// TIA Portal V16 export
// export: Created 2022-11-17T15:49:39.066239Z, ExportSetting WithDefaults, DisplayName Totally Integrated Automation Portal, DisplayVersion V16 Update 6, DisplayName TIA Portal Version Control Interface, DisplayVersion V16 Update 2, DisplayName TIA Portal Openness, DisplayVersion V16 Update 6, DisplayName SINAMICS Startdrive Advanced, DisplayVersion V16 Update 5, DisplayName SINAMICS Startdrive G130, G150, S120, S150, SINAMICS MV, S210, DisplayVersion V16 Update 5, DisplayName SINAMICS Startdrive G110M, G120, G120C, G120D, G120P, G115D, DisplayVersion V16 Update 5, DisplayName STEP 7 Professional, DisplayVersion V16 Update 6, DisplayName STEP 7 Safety, DisplayVersion V16, DisplayName WinCC Advanced, DisplayVersion V16 Update 6
DATA_BLOCK "DB20_DisplaySysdata"   // DB20
{ S7_Optimized_Access := 'FALSE' }
AUTHOR : Robopac
VERSION : 0.0
// stored: AutoNumber false, IsOnlyStoredInLoadMemory false, IsWriteProtectedInAS false
   VAR RETAIN
      dbd0 : DInt := 238;   // Step for encoder spool carriage movement (mm/100) (Display-Sysadata)
      dbw4 : Int := 6;   // Histeresys for spool carriage positioning (mm) (Display-Sysdata)
      dbw6 : Int := 50;   // Deceleration for spool carriage positioning (mm) (Display-Sysdata)
      dbw8 : Int := 50;   // Low speed for spool carriage movement (%) (Display-Sysdata)
      dbw10 : Int := 100;   // High speed for spool carriage movement (%) (Display-Sysdata)
      dbw12 : Int := 430;   // Spool height (mm) (Display-Sysdata)
      dbw14 : Int := 0;   // Spool carriage down position (mm) (Display-Sysadata)
      dbw16 : Int := 100;   // First step speed for spool carriage movement (%) (Display-Sysadata)
      dbw18 : Int := 240;   // Offset for ftc pallet height (mm) (Display-Sysdata)
      dbw20 : Int := 180;   // Pressure plate height (mm) (Display-Sysdata)
      dbw22 : Int := 7;   // Distance lifter up - conveyor (mm) (Display-Sysdata)
      dbw24 : Int := 0;   // Spool carriage height for film broken cycle (mm) (Display-Sysdata)
      dbw26 : Int := 50;   // Low speed angle to stop rotation (Display-Sysdata)
      dbw28 : Int := 1000;   // Jog1 speed for fast prestretch rool (Display-Sysadata)
      dbw30 : Int := 45;   // Offset for SCSP/2 (Display-Sysadata)
      dbw32 : Int := 78;
      dbw34 : Int := 1100;   // Arm rotation motor and gearbox type (Display-Sysdata)
      dbw36 : Int := 0;   // Delay for test cycle (Display-Sysdata)
      dbx38_0 : Bool := FALSE;   // Film ended or broken cycle included/excluded(1) (Display-Sysdata)
      dbx38_1 : Bool := FALSE;   // Conveyor encoder alarm included(0)/excluded (Display-Sysdata)
      dbx38_2 : Bool := FALSE;   // Test cycle included(1)/excluded (Display-Sysdata)
      dbx38_3 : Bool := FALSE;   // Top film ended or broken included(0)/excluded (Display-Sysdata)
      dbx38_4 : Bool := TRUE;   // Pallet height with pressure plate priority (Display-Sysdata)
      dbx38_5 : Bool := TRUE;   // Spool carriage upward during arm deceleration excluded/included(1) (Display-Sys
      dbx38_6 : Bool := FALSE;   // Pressure plate upward before(0)/after cut cycle (Display-Sysdata)
      dbx38_7 : Bool := FALSE;   // Bit stop pallet infeed (Display-Sysdata)
      dbx39_0 : Bool := FALSE;   // Timeout included/excluded(1) (Display-Sysdata)
      dbx39_1 : Bool := FALSE;   // Reverse cycle request from hmi (Display-Main page)
      dbx39_2 : Bool := FALSE;
      dbx39_3 : Bool := FALSE;
      dbx39_4 : Bool := FALSE;
      dbx39_5 : Bool := FALSE;
      dbx39_6 : Bool := TRUE;   // Top fast cycle
      dbx39_7 : Bool := FALSE;
      dbw40 : Int := 65;   // Spool carriage upward during arm deceleration (mm) (Display-Sysdata)
      dbw42 : Int := 1360;   // Step for infeed conveyor encoder (mm/100) (Display-Sysdata)
      dbw44 : Int := -210;   // Pulse offset for rotation encoder (Display-Sysdata)
      dbw46 : Int := 0;   // Pallet lenght for small pallet (Display-Sysdata)
      dbw48 : Int := 0;   // Decentering for pallet positioning (Display-Sysdata)
      dbw50 : Int := 500;   // Quote for airblower on (mm) (Display-Sysdata)
      dbw52 : Int := 0;   // Spool carriage up to cover film tail (Display-Sysdata)
      dbw54 : Int := 3000;   // Cutting time (Display-Sysdata)
      dbw56 : Int := 1500;   // MAX TIRO SU CELLA (kg) [ex SysdataTempoTwist]
      dbw58 : Int := 2400;   // Delay to open clamp (Display-Sysdata)
      dbw60 : Int := 0;   // Table rotation clampcut phase (°) (Display-Sysdata)
      dbw62 : Int := 200;   // Quote to open clamp (Display-Sysdata)
      dbw64 : Int := 0;   // Step for top carriage forward/backward (mm/100) (Display-Sysdata)
      dbw66 : Int := 1000;   // Step for top carriage upward/downward (mm/100) (Display-Sysdata)
      dbw68 : Int := 600;   // Deceleration for top carriage forward/backward (Display-Sysdata)
      dbw70 : Int := 1500;   // Top carriage up position (Display-Sysdata)
      dbw72 : Int := 0;   // Spool carriage position for top cycle (Display-Sysdata)
      dbw74 : Int := 0;   // Delay for spool carriage downward during top cycle (Display-Sysdata)
      dbw76 : Int := 0;   // Tabke rotation load phase (°) (Display-Sysdata)
      dbw78 : Int := 0;   // Table rotation unload phase (°) (Display-Sysdata)
      dbd80 : DInt := 5627;   // Step for encoder table rotation movement (°/p) (Display-Sysdata)
      dbw84 : Int := 18;   // Histeresys for table rotation positioning (°) (Display-Sysdata)
      dbw86 : Int := 2100;   // Deceleration for table rotation positioning (Hz/sec) (Display-Sysdata)
      dbw88 : Int := 10;   // Low speed for table rotation movement (%) (Display-Sysdata)
      dbw90 : Int := 100;   // High speed for table rotation movement (%) (Display-Sysdata)
      dbw92 : Int := 1800;   // Delay to stop top carriage forward for top film broken
      dbw94 : Int := 1000;   // Delay for top pallet height reading photocell (fast cycle)
      dbw96 : Int := 60;
      dbw98 : Int := 20;
   END_VAR
BEGIN
END_DATA_BLOCK
